{attribute 'qualified_only'}
VAR_GLOBAL
    fbArbiter: FB_Arbiter;
    fbFastFaultOutput1: FB_HardwareFFOutput;
    fbFastFaultOutput2: FB_HardwareFFOutput;
END_VAR

(* stored: Version 1.1.0.1, ProductVersion 3.1.4022.12
   GVL PMPS: Id {53ff6662-fc6b-4a00-9f46-186d8230905b} *)
